// TIA Portal V17 export
// export: Created 2023-12-22T15:03:03.3337934Z, ExportSetting WithDefaults, DisplayName Totally Integrated Automation Portal, DisplayVersion V17, DisplayName TIA Portal Openness, DisplayVersion V17, DisplayName TIA Portal Version Control Interface, DisplayVersion V17, DisplayName STEP 7 Professional, DisplayVersion V17, DisplayName STEP 7 Safety, DisplayVersion V17, DisplayName WinCC Advanced, DisplayVersion V17
DATA_BLOCK "DOx_1_DB"   // DB210
VERSION : 0.1
// stored: AutoNumber false, DBAccessibleFromOPCUA true, DBAccessibleFromWebserver true, InstanceOfName DOx_1, InstanceOfType FB
"DOx_1"
   // VAR RETAIN
   //    All_Alarm { S7_SetPoint := 'True'} : "DO_ex";
   //    command_2 { S7_SetPoint := 'True'} : "DO_ex";
   //    command_3 { S7_SetPoint := 'True'} : "DO_ex";
   //    command_4 { S7_SetPoint := 'True'} : "DO_ex";
   //    command_5 { S7_SetPoint := 'True'} : "DO_ex";
   //    command_6 { S7_SetPoint := 'True'} : "DO_ex";
   //    command_7 { S7_SetPoint := 'True'} : "DO_ex";
   //    command_8 { S7_SetPoint := 'True'} : "DO_ex";
   //    command_9 { S7_SetPoint := 'True'} : "DO_ex";
   //    command_10 { S7_SetPoint := 'True'} : "DO_ex";
   //    command_11 { S7_SetPoint := 'True'} : "DO_ex";
   //    command_12 { S7_SetPoint := 'True'} : "DO_ex";
   //    Time_DTL { S7_SetPoint := 'True'} : DTL := DTL#2023-05-02-18:36:48.708907168;
   // END_VAR
BEGIN
   All_Alarm.Use.Inverse := FALSE;
   All_Alarm.Use.Indirect := TRUE;
   All_Alarm.Use.Impulse := FALSE;
   All_Alarm.ADDR_Byte := 0;
   All_Alarm.ADDR_Bit := 1;
   All_Alarm.T_Impulse.SP := 16#02;
   command_2.Use.Inverse := FALSE;
   command_2.Use.Indirect := TRUE;
   command_2.Use.Impulse := FALSE;
   command_2.ADDR_Byte := 0;
   command_2.ADDR_Bit := 9;
   command_2.T_Impulse.SP := 16#02;
   command_3.Use.Inverse := FALSE;
   command_3.Use.Indirect := TRUE;
   command_3.Use.Impulse := FALSE;
   command_3.ADDR_Byte := 0;
   command_3.ADDR_Bit := 9;
   command_3.T_Impulse.SP := 16#02;
   command_4.Use.Inverse := FALSE;
   command_4.Use.Indirect := TRUE;
   command_4.Use.Impulse := FALSE;
   command_4.ADDR_Byte := 0;
   command_4.ADDR_Bit := 9;
   command_4.T_Impulse.SP := 16#02;
   command_5.Use.Inverse := FALSE;
   command_5.Use.Indirect := TRUE;
   command_5.Use.Impulse := FALSE;
   command_5.ADDR_Byte := 0;
   command_5.ADDR_Bit := 9;
   command_5.T_Impulse.SP := 16#02;
   command_6.Use.Inverse := FALSE;
   command_6.Use.Indirect := TRUE;
   command_6.Use.Impulse := FALSE;
   command_6.ADDR_Byte := 0;
   command_6.ADDR_Bit := 9;
   command_6.T_Impulse.SP := 16#02;
   command_7.Use.Inverse := FALSE;
   command_7.Use.Indirect := TRUE;
   command_7.Use.Impulse := FALSE;
   command_7.ADDR_Byte := 0;
   command_7.ADDR_Bit := 9;
   command_7.T_Impulse.SP := 16#02;
   command_8.Use.Inverse := FALSE;
   command_8.Use.Indirect := TRUE;
   command_8.Use.Impulse := FALSE;
   command_8.ADDR_Byte := 0;
   command_8.ADDR_Bit := 9;
   command_8.T_Impulse.SP := 16#02;
   command_9.Use.Inverse := FALSE;
   command_9.Use.Indirect := TRUE;
   command_9.Use.Impulse := FALSE;
   command_9.ADDR_Byte := 0;
   command_9.ADDR_Bit := 9;
   command_9.T_Impulse.SP := 16#02;
   command_10.Use.Inverse := FALSE;
   command_10.Use.Indirect := TRUE;
   command_10.Use.Impulse := FALSE;
   command_10.ADDR_Byte := 0;
   command_10.ADDR_Bit := 9;
   command_10.T_Impulse.SP := 16#02;
   command_11.Use.Inverse := FALSE;
   command_11.Use.Indirect := TRUE;
   command_11.Use.Impulse := FALSE;
   command_11.ADDR_Byte := 0;
   command_11.ADDR_Bit := 9;
   command_11.T_Impulse.SP := 16#02;
   command_12.Use.Inverse := FALSE;
   command_12.Use.Indirect := TRUE;
   command_12.Use.Impulse := FALSE;
   command_12.ADDR_Byte := 0;
   command_12.ADDR_Bit := 9;
   command_12.T_Impulse.SP := 16#02;
END_DATA_BLOCK
